TYPE DUT_stDeleteBatchToProductionQueue :
STRUCT
	return_			: DINT;
	BatchId	: STRING(50);
END_STRUCT
END_TYPE

(* stored: Version 1.1.0.1, ProductVersion 3.1.4024.15
   DUT DUT_stDeleteBatchToProductionQueue: Id {f2ffa58b-0093-4d82-b535-0bc499b2ea8a} *)
